RoboDK station: dance_sim.rdk

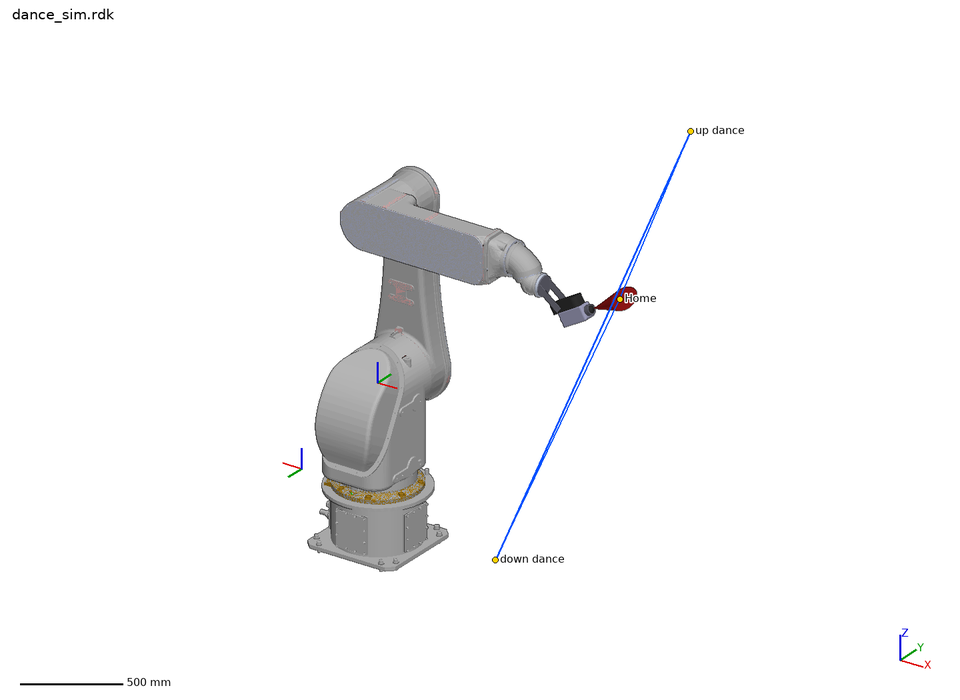
[picture v0: the station drawn from its stored meshes, robots at their saved joint values, targets as dots, program paths as lines]
Station dance_sim (saved by RoboDK 5.5.4). Poses are relative to the parent item; angles as X-Y-Z fixed-axis rotations.
Station parameters (name, value as stored): LIN64
  - frame Fanuc P-50iB/10L Base at (0, 0, 987.61) mm
    - robot Fanuc P-50iB/10L: 6 axes, payload 10 kg, reach 1800 mm, repeatability 0.2 mm, weight 331 kg
        modified DH rows (alpha deg, a mm, theta deg, d mm): 0, 0, 0, 850; -90, 0, -90, 0; 0, 900, 0, 0; -90, 0, -90, 863.603; 70, 0, 0, 106.418; -70, 0, 0, 82
        base shift (0, 0, -850) mm
        joint limits [-160, -45, -205, -360, -360, -360] to [160, 120, 165, 360, 360, 360]; home [0, 0, 0, 0, 0, 0]; saved at [0, 0, 0, 0, 0, 0]
      - tool Paint gun, TCP at (50, 0, 450) mm, rotated rx 0 ry 30 rz 0 deg, size 203.2 x 279.7 x 471.5 mm
  - frame Frame 2 at (-800, 500, 100) mm, rotated rx 0 ry 0 rz 180 deg
    - target Home (Cartesian target) at (-2232, 500, 1737.61) mm, rotated rx 0 ry -60 rz 0 deg; joints [0, 0, 0, 0, 0, 0] of Fanuc P-50iB/10L
    - target down dance (Cartesian target) at (-2056.09, 1299.2, 600.31) mm, rotated rx 0 ry -60 rz 0 deg; joints [-51.977, 56.044, -64.639, -51.372, 80.426, 53.396] of Fanuc P-50iB/10L
    - target up dance (Cartesian target) at (-2056.09, -352.75, 2255.64) mm, rotated rx 0 ry -60 rz 0 deg; joints [52.315, 23.559, 27.618, -211.149, 61.253, 202.023] of Fanuc P-50iB/10L
  - program dance (8 instructions, listed below)
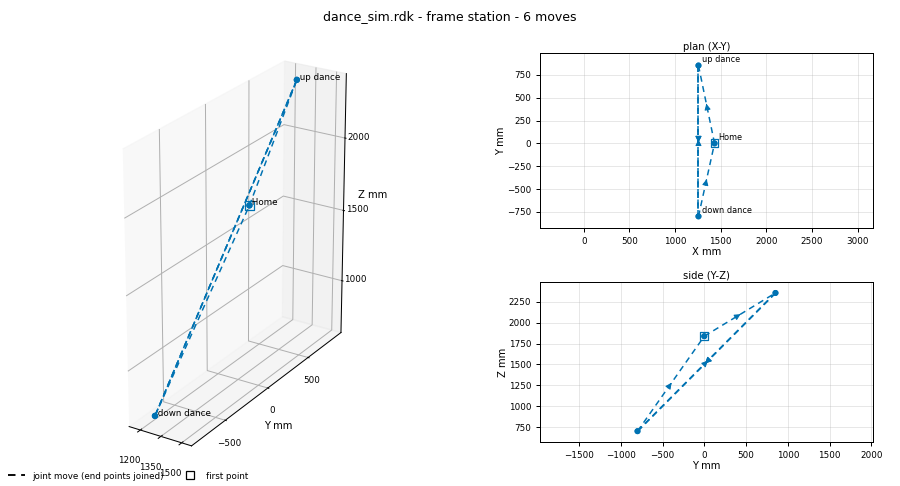
[picture p0: tool path of dance_sim.rdk in frame station, 6 of 6 moves have a stored position in this frame; points joined in program order, loops and branches not executed]

--- program dance (robot Fanuc P-50iB/10L) ---
  Set Ref.: Frame 2
  Set Tool: Paint gun
  MoveJ (Home)
  MoveJ (up dance)
  MoveJ (down dance)
  MoveJ (up dance)
  MoveJ (down dance)
  MoveJ (Home)
